// TwinCAT 3 PLC project PLCStudent
// ProgramVersion: 3.1.4022.4
// libraries:
//   Tc2_Standard, * (Beckhoff Automation GmbH)
//   Tc2_System, * (Beckhoff Automation GmbH)
//   Tc3_Module, * (Beckhoff Automation GmbH)
//   VisuSymbols,3.5.10.0,System
// project tree:
//   / GlobalTextList.TcGTLO, PlcTask.TcTTO, Visualization Manager.TcVMO (not stored)
//   GVLs/ GVL.TcGVL
//   POUs/ FB_PositionDisplay.TcPOU, MAIN.TcPOU, SFC.TcPOU
//   VISUs/ Display.TcIPO (not stored), HMIoperator.TcVIS

CONFIGURATION PLCStudent
    RESOURCE PLC ON TwinCAT3
        TASK PlcTask(INTERVAL := T#20ms, PRIORITY := 20);
        PROGRAM MAIN WITH PlcTask : MAIN;
    END_RESOURCE
END_CONFIGURATION

// ---- GVLs/GVL.TcGVL
{attribute 'qualified_only'}
VAR_GLOBAL
//Input to PLC from process
	ixAGVStrobe		AT %I*:	BOOL;	(* AGV strobe signal *)
	iiAtPos			AT %I*:	INT;	(* Actual position of AGV *)
	qxStartButton   AT %Q*: BOOL;   (* Start Button*)
	qxStopButton    AT %Q*: BOOL;   (* Stop Button*)
	qxResetButton   AT %Q*: BOOL;   (* Reset Button*)
	
//Output from PLC to process
	qxPLCStrobe		AT %Q*:	BOOL;	(* PLC strobe signal *)
	qiGotoPos		AT %Q*:	INT;	(* Target position for AGV *)

// Additional global variables
	ixAGVMoving     AT %I*: BOOL;   (* AGV Moving*)
	ixAGVLoc        AT %I*: STRING; (* AGV Location*)
END_VAR

// ---- POUs/MAIN.TcPOU
PROGRAM MAIN
VAR
END_VAR

SFC();

END_PROGRAM

// ---- POUs/SFC.TcPOU
PROGRAM SFC
VAR
	Target: ARRAY [1..5] OF STRING := ['HOME','PosA','PosB','PosC','PosD'];
    TargIndex: INT:=0;
	qxGreenLamp :BOOL;
	qxRedLamp :BOOL;
	ElepseTime : TIME;
	TON_Blink1: TON;
	TON_Blink0: TON;
	Invisible: BOOL;
	MovingLamp: BOOL;
	ResetMemory : BOOl;
	TON_Moving: TON;
END_VAR

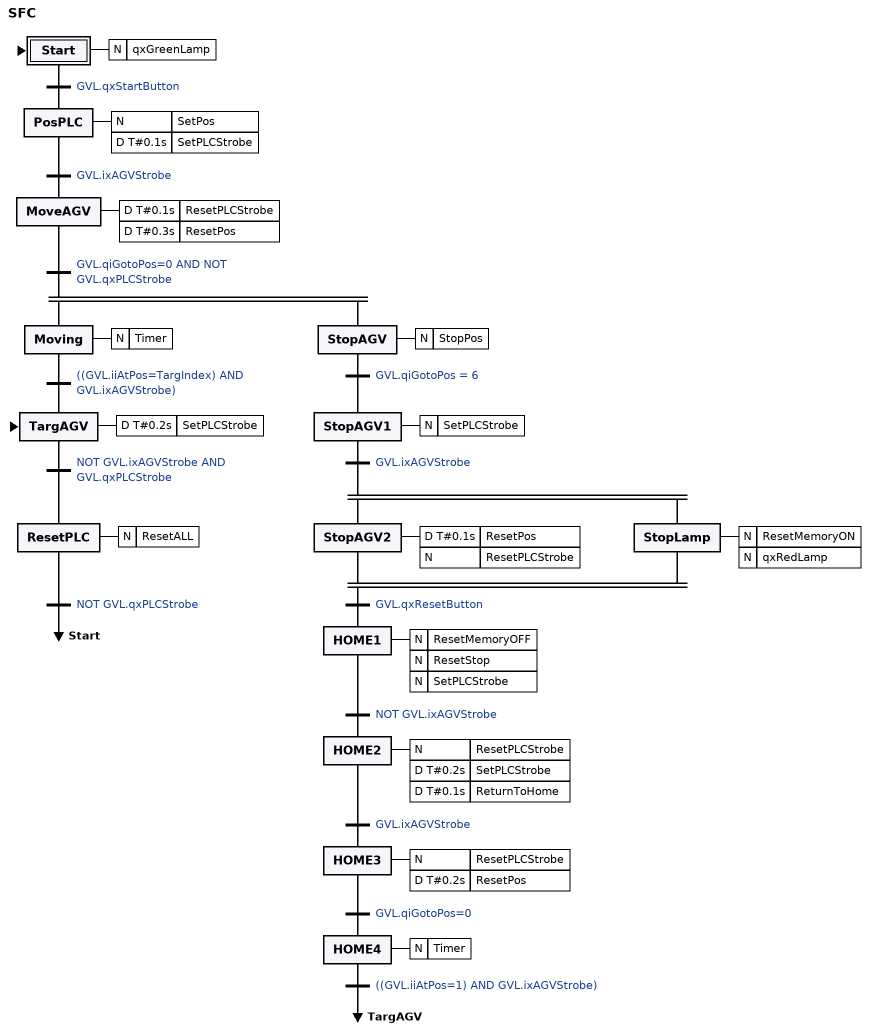
INITIAL_STEP Start:
    qxGreenLamp(N);
END_STEP
TRANSITION FROM Start TO PosPLC
    := GVL.qxStartButton;
END_TRANSITION
STEP PosPLC:
    SetPos(N);
    SetPLCStrobe(D, T#0.1s);
END_STEP
TRANSITION FROM PosPLC TO MoveAGV
    := GVL.ixAGVStrobe;
END_TRANSITION
STEP MoveAGV:
    ResetPLCStrobe(D, T#0.1s);
    ResetPos(D, T#0.3s);
END_STEP
TRANSITION FROM MoveAGV TO (Moving, StopAGV)
    := GVL.qiGotoPos=0 AND NOT GVL.qxPLCStrobe;
END_TRANSITION
STEP Moving:
    Timer(N);
END_STEP
STEP StopAGV:
    StopPos(N);
END_STEP
TRANSITION FROM StopAGV TO StopAGV1
    := GVL.qiGotoPos = 6;
END_TRANSITION
STEP StopAGV1:
    SetPLCStrobe(N);
END_STEP
TRANSITION FROM StopAGV1 TO (StopAGV2, StopLamp)
    := GVL.ixAGVStrobe;
END_TRANSITION
STEP StopAGV2:
    ResetPos(D, T#0.1s);
    ResetPLCStrobe(N);
END_STEP
STEP StopLamp:
    ResetMemoryON(N);
    qxRedLamp(N);
END_STEP
TRANSITION FROM (StopAGV2, StopLamp) TO HOME1
    := GVL.qxResetButton;
END_TRANSITION
STEP HOME1:
    ResetMemoryOFF(N);
    ResetStop(N);
    SetPLCStrobe(N);
END_STEP
TRANSITION FROM HOME1 TO HOME2
    := NOT GVL.ixAGVStrobe;
END_TRANSITION
STEP HOME2:
    ResetPLCStrobe(N);
    SetPLCStrobe(D, T#0.2s);
    ReturnToHome(D, T#0.1s);
END_STEP
TRANSITION FROM HOME2 TO HOME3
    := GVL.ixAGVStrobe;
END_TRANSITION
STEP HOME3:
    ResetPLCStrobe(N);
    ResetPos(D, T#0.2s);
END_STEP
TRANSITION FROM HOME3 TO HOME4
    := GVL.qiGotoPos=0;
END_TRANSITION
STEP HOME4:
    Timer(N);
END_STEP
TRANSITION FROM HOME4 TO TargAGV
    := ((GVL.iiAtPos=1) AND GVL.ixAGVStrobe);
END_TRANSITION
TRANSITION FROM Moving TO TargAGV
    := ((GVL.iiAtPos=TargIndex) AND GVL.ixAGVStrobe);
END_TRANSITION
STEP TargAGV:
    SetPLCStrobe(D, T#0.2s);
END_STEP
TRANSITION FROM TargAGV TO ResetPLC
    := NOT GVL.ixAGVStrobe AND GVL.qxPLCStrobe;
END_TRANSITION
STEP ResetPLC:
    ResetALL(N);
END_STEP
TRANSITION FROM ResetPLC TO Start
    := NOT GVL.qxPLCStrobe;
END_TRANSITION
// branch label Stop
// branch label MoveB

ACTION ResetALL:
GVL.qxPLCStrobe := FALSE;
GVL.qxStartButton := FALSE;
GVL.qxResetButton := FALSE;
GVL.qxStopButton := FALSE;
END_ACTION

ACTION ResetMemoryOFF:
ResetMemory := FALSE;
END_ACTION

ACTION ResetMemoryON:

ResetMemory := TRUE ;
END_ACTION

ACTION ResetPLCStrobe:
GVL.qxPLCStrobe := FALSE;
END_ACTION

ACTION ResetPos:
Gvl.qiGotoPos := 0;
END_ACTION

ACTION ResetStart:
GVL.qxStartButton :=FALSE;
END_ACTION

ACTION ResetStop:
GVL.qxStopButton := FALSE;
END_ACTION

ACTION ResetTarg:
TargIndex :=0;
END_ACTION

ACTION ReturnToHome:
GVL.qiGotoPos := 1;
GVL.qxResetButton := FALSE;
END_ACTION

ACTION SetPLCStrobe:
GVL.qxPLCStrobe := TRUE;
END_ACTION

ACTION SetPos:
GVL.qiGotoPos := TargIndex;
GVL.qxStartButton := FALSE;
END_ACTION

ACTION StopPos:
IF GVL.qxStopButton THEN
	GVL.qiGotoPos := 6;
END_IF
END_ACTION

ACTION Timer:
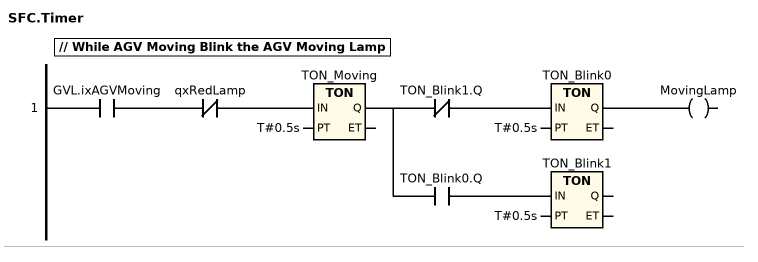
// NETWORK 1
// label: // While AGV Moving Blink the AGV Moving Lamp
TON_Moving(IN := GVL.ixAGVMoving AND NOT qxRedLamp, PT := T#0.5s); // TON
TON_Blink0(IN := TON_Moving.Q AND NOT TON_Blink1.Q, PT := T#0.5s); // TON
MovingLamp := TON_Blink0.Q;
TON_Blink1(IN := TON_Moving.Q AND TON_Blink0.Q, PT := T#0.5s); // TON
END_ACTION

END_PROGRAM

// ---- POUs/FB_PositionDisplay.TcPOU
FUNCTION_BLOCK FB_PositionDisplay
VAR_INPUT
	Position : STRING;
END_VAR
VAR_OUTPUT
	ixDisplay : INT;
END_VAR
VAR
END_VAR

IF Position = 'HOME' THEN
	ixDisplay := 1;
ELSIF Position  = 'Pos A' THEN
	ixDisplay := 2;
ELSIF Position  = 'Pos B' THEN
	ixDisplay := 3;
ELSIF Position  = 'Pos C' THEN
	ixDisplay := 4;
ELSIF Position  = 'Pos D' THEN
	ixDisplay := 5;
ELSE
	ixDisplay := 0;
END_IF

END_FUNCTION_BLOCK

// ---- GlobalTextList.TcGTLO
TEXTLIST GlobalTextList
  532 = 'AGV Moving'
  272 = 'Display'
  574 = 'Pos %i '
  173 = 'Ready'
  82 = 'Reset'
  965 = 'Select Target'
  689 = 'STARt'
  610 = 'START'
  758 = 'Start'
  259 = 'Stop'
  946 = 'Stop Lamp'
END_TEXTLIST

// ---- VISUs/HMIoperator.TcVIS
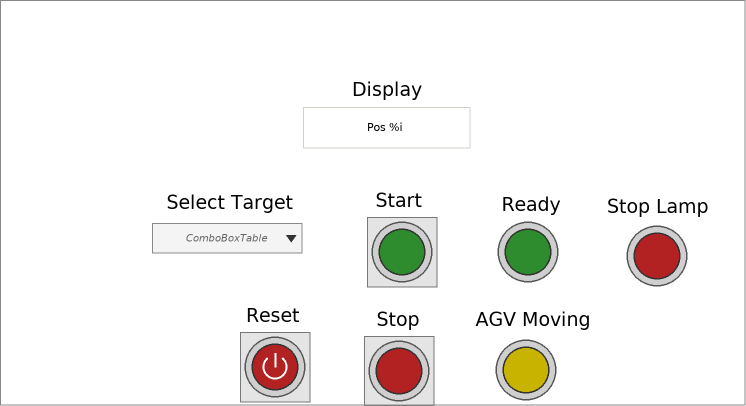
VISUALIZATION HMIoperator  // 746x406, background image Display.Display
    PowerSwitch (240,332 70x70), variable: GVL.qxResetButton, input disabled if: NOT SFC.ResetMemory, behaviour: TOGGLE, style: Switch-PowerSwitch-Red
    PushSwitchLed (367,217 70x70), variable: GVL.qxStartButton, input disabled if: GVL.ixAGVMoving, behaviour: TOGGLE, style: Switch-PushSwitchLed-Green
    PushSwitchLed (364,336 70x70), variable: GVL.qxStopButton, input disabled if: NOT GVL.ixAGVMoving, behaviour: TOGGLE, style: Switch-PushSwitchLed-Red
    ComboBoxTable (152,223 150x30), variable: SFC.TargIndex, input disabled if: GVL.ixAGVMoving, data array: SFC.Target
        p3854506369: SFC.Target[INDEX]
    Lamp1 (493,217 70x70), variable: SFC.qxGreenLamp, style: Lamp-Lamp1-Green
    Textfield (303,107 167x41), "Pos %i", text variable: GVL.iiAtPos, invisible if: GVL.ixAGVMoving
    Rectangle (142,189 176x27), "Select Target"
    Rectangle (570,193 176x27), "Stop Lamp"
    Rectangle (445,306 176x27), "AGV Moving"
    Lamp1 (491,335 70x70), variable: SFC.MovingLamp, style: Lamp-Lamp1-Yellow
    Rectangle (352,186 94x29), "Start"
    Rectangle (351,305 94x29), "Stop"
    Rectangle (226,301 94x29), "Reset"
    Rectangle (299,76 176x27), "Display"
    Lamp1 (622,221 70x70), variable: SFC.qxRedLamp, style: Lamp-Lamp1-Red
    Rectangle (443,191 176x27), "Ready"
END_VISUALIZATION
